{attribute 'linkalways'} 
{attribute 'no_explicit_call' := 'This FB is a CLASS and must be accessed using methods or properties'}
{attribute 'enable_dynamic_creation'}
FUNCTION_BLOCK _TcVnVector3_LREAL EXTENDS AliasDatatypeBase
VAR
	localData : TcVnVector3_LREAL;
	activeData : REFERENCE TO TcVnVector3_LREAL REF= localData;
	aliasBaseDatatype : _Array0to2OfLREAL;
END_VAR

PROPERTY PUBLIC Address : PVOID
GET
Address := ADR(activeData);
END_GET
END_PROPERTY

METHOD PUBLIC ClearReference
VAR_INPUT
END_VAR
activeData REF= localData;
SetBaseDatatypeReference();
END_METHOD

METHOD PUBLIC Clone : I_Datatype
VAR
    pClone : POINTER TO _TcVnVector3_LREAL;
END_VAR
pClone := __NEW(_TcVnVector3_LREAL);
Clone := pClone^;
END_METHOD

METHOD FB_init : BOOL
VAR_INPUT
	bInitRetains : BOOL; // if TRUE, the retain variables are initialized (warm start / cold start)
	bInCopyCode : BOOL;  // if TRUE, the instance afterwards gets moved into the copy code (online change)
	//InitialValue : <type>; // if possible, not all values can be initialized
END_VAR
//localData := InitialValue; // if possible, not all values can be initialized
SetBaseDatatypeReference();
AddBaseDatatype(aliasBaseDatatype);
END_METHOD

PROPERTY PUBLIC Identifier : T_MAXSTRING
GET
Identifier := 'TcVnVector3_LREAL';
END_GET
END_PROPERTY

METHOD PUBLIC MakeReferenceTo
VAR_INPUT
	ReferenceTarget : REFERENCE TO TcVnVector3_LREAL;
END_VAR
activeData REF= ReferenceTarget;
SetBaseDatatypeReference();
END_METHOD

METHOD PROTECTED SetBaseDatatypeReference
VAR_INPUT
END_VAR
aliasBaseDatatype.MakeReferenceTo(activeData);
END_METHOD

PROPERTY PUBLIC Size : UDINT
GET
Size := SIZEOF(activeData);
END_GET
END_PROPERTY

METHOD TryMakeReferenceTo : BOOL
VAR_INPUT
	Target : I_Datatype;
END_VAR
VAR
	pTargetData : POINTER TO TcVnVector3_LREAL;
END_VAR
IF NOT IsEquivalentTo(Target) THEN
	RETURN;
END_IF

pTargetData := Target.Address;
activeData REF= pTargetData^;
SetBaseDatatypeReference();
TryMakeReferenceTo := TRUE;
END_METHOD

PROPERTY PUBLIC Value : REFERENCE TO TcVnVector3_LREAL
GET
Value REF= activeData;
END_GET
END_PROPERTY

END_FUNCTION_BLOCK

(* stored: Version 1.1.0.1, ProductVersion 3.1.4024.13
   POU _TcVnVector3_LREAL: Id {3b3acf8d-0ced-02eb-192a-08578e76ce3f}, SpecialFunc None
   Folder Core: Id {af9e7799-40ba-0909-1ba3-b8adbd4bafa2}
   Folder Protected: Id {a3175121-480b-0298-3875-5019fa34e3d5}
   Folder Customize: Id {dbb8a646-2622-0734-2b55-3b67d08febb3}
   Folder Constructor: Id {58d5e5e2-562c-0e92-2c05-fb484f751292}
   Property Address: Id {cad3dcd8-28e4-0dd1-2598-9c0ccf63b33b}
   Get Get: Id {5c2241b8-2ce8-016e-139a-9013cc4d0f34}
   Method ClearReference: Id {53518119-c45f-00d6-1ad3-cc4a5e54696d}
   Method Clone: Id {dffaad20-d445-032f-1c25-cc3e1ec3afc7}
   Method FB_init: Id {96bba5eb-d565-07e2-0527-eee58896b04e}
   Property Identifier: Id {d55a7b79-ffe7-07e6-37bf-49a346575014}
   Get Get: Id {1b8eab33-ba39-0006-3a00-daddd61dae1d}
   Method MakeReferenceTo: Id {29af583d-1358-0de9-2b1a-e579b32b3937}
   Method SetBaseDatatypeReference: Id {8801c6ce-14cf-007f-2755-d253e58dc76c}
   Property Size: Id {7bd5b0d5-5573-0788-07b4-ad70d0c44d34}
   Get Get: Id {2e82a136-83d2-0bb7-3e87-7859c2a1668a}
   Method TryMakeReferenceTo: Id {f8c44f30-468b-0950-2a11-472d0c5f6894}
   Property Value: Id {0e2e3e6b-e74e-0146-1f3b-2f7c7ad24df1}
   Get Get: Id {c1e8d4a4-1986-089e-1588-dd67a62bde10} *)
